FUNCTION_BLOCK FB_CycleTrigger // This function can be used to start state machines and wait for them to finish
VAR_OUTPUT
	bStart 	: BOOL ; // Start cycle 
	bBusy 	: BOOL ; // cycle is bussy
	bDone	: BOOL ; // cycle is done
END_VAR
VAR
	fbreStartCycle : R_TRIG ; // rising edge trigger for cycle start
END_VAR

ACTION Reset:
bDone 	:= FALSE;
bBusy 	:= FALSE;
bStart	:= FALSE;
END_ACTION

ACTION SetDone:
bBusy := FALSE 	;
bDone := TRUE	;
END_ACTION

ACTION SetStart:
IF fbreStartCycle.Q THEN
	bBusy := TRUE; 
ELSIF bDone THEN 
	bStart := FALSE;
ELSE
	bStart := TRUE;
END_IF

fbreStartCycle(CLK := bStart);
END_ACTION

END_FUNCTION_BLOCK

(* stored: Version 1.1.0.1, ProductVersion 3.1.4024.11
   POU FB_CycleTrigger: Id {3ee0d948-25d9-4a8a-a0c3-91cb3bb1b3ed}, SpecialFunc None
   Action Reset: Id {2e606475-f64a-48b1-ba1f-3b3677d1e9ec}
   Action SetDone: Id {6d335d99-9d45-408a-9374-5d527d113da7}
   Action SetStart: Id {ca054a1f-b63d-4ae6-9552-74e489f45e0b} *)
